Fanuc KAREL source: ko00006.KL

PROGRAM KO00006
%STACKSIZE=65535
%PRIORITY=65535
%NOLOCKGROUP
VAR
P1 : POSITION
P2 : POSITION
P3 : POSITION
P4 : POSITION
OUT : XYZWPR
BEGIN
-- UNRESOLVED_PC line 10 opcodes [27 22 1C 22 1C 22 1C 22 1C 76 7E 4A] marker_code=0
END KO00006
